RoboDK station: Assistive_UR5e.rdk

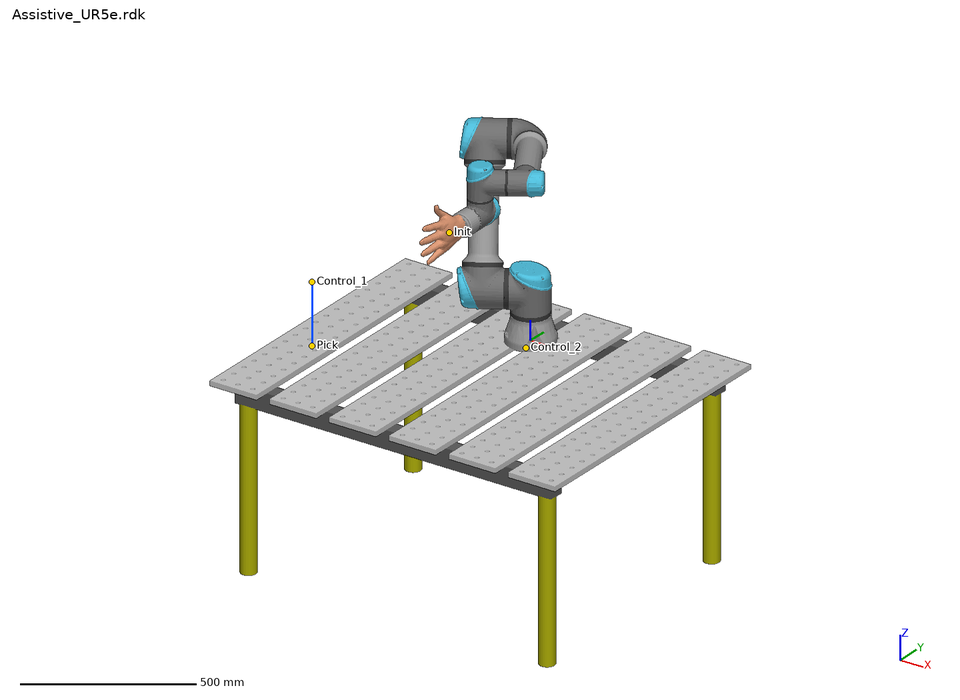
[picture v0: the station drawn from its stored meshes, robots at their saved joint values, targets as dots, program paths as lines]
Station Assistive_UR5e_SW (saved by RoboDK 5.9.2). Poses are relative to the parent item; angles as X-Y-Z fixed-axis rotations.
  - frame UR5e Base at (0, 0, 0) mm
    - robot UR5e: 6 axes, payload 5 kg, reach 850 mm, repeatability 0.03 mm, weight 18.4 kg
        modified DH rows (alpha deg, a mm, theta deg, d mm): 0, 0, 0, 162.5; 90, 0, 180, 0; 0, 425, 0, 0; 0, 392.25, 0, 133.3; -90, 0, 0, 99.7; 90, 0, 180, 99.6
        joint limits [-360, -360, -360, -360, -360, -360] to [360, 360, 360, 360, 360, 360]; home [0, -90, -90, 0, 90, 0]; saved at [-57.836, -65.392, -107.167, 172.559, -57.836, 0]
      - tool Hand, TCP at (0, 0, 50) mm, size 54.8 x 155.9 x 193.5 mm, geometry from Hand.stl
  - frame World at (0, 0, 0) mm
    - object Table at (0, 0, 0) mm, size 1193.8 x 965.2 x 609.6 mm, geometry from welding_table.sld
    - target Init (Cartesian target) at (0, -400, 500) mm, rotated rx 90 ry 0 rz 0 deg; joints [-57.836, -65.392, -107.167, 172.559, -57.836, 0] of UR5e
    - target Control_1 (joint target) at (-370, -550, 300) mm, rotated rx 90 ry -85.28 rz 0 deg; joints [-118.588, -113.226, -89.788, -156.986, -118.588, 85.275] of UR5e
    - target Pick (joint target) at (-370, -550, 100) mm, rotated rx 90.01 ry -85.28 rz -0.01 deg; joints [-118.588, -129.044, -99.259, -131.698, -118.588, 85.275] of UR5e
    - target Control_2 (joint target) at (370, -550, 300) mm, rotated rx 90.01 ry -85.28 rz -0.01 deg; joints [-33.107, -113.226, -89.788, -156.987, -33.108, 85.277] of UR5e
    - target Show (joint target) at (370, -550, 300) mm, rotated rx 90.01 ry 87.37 rz 0.01 deg; joints [-33.107, -113.226, -89.788, -156.987, -33.108, -87.373] of UR5e
  - program Init (3 instructions, listed below)
  - program Pick_object (6 instructions, listed below)
  - program Show_object (4 instructions, listed below)
  - program MainProgram (4 instructions, listed below)
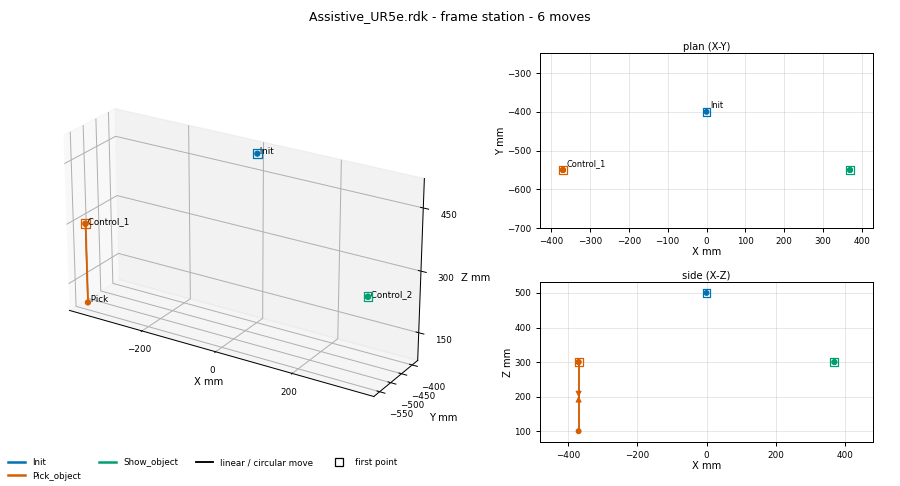
[picture p0: tool path of Assistive_UR5e.rdk in frame station, 6 of 6 moves have a stored position in this frame; points joined in program order, loops and branches not executed]

--- program Init (robot UR5e) ---
  Est. Ref.: UR5e Base
  Est. herr: Hand
  MoveJ (Init)

--- program Pick_object (robot UR5e) ---
  Est. Ref.: UR5e Base
  Est. herr: Hand
  MoveL (Control_1)
  MoveL (Pick)
  Pausa 1.0 s
  MoveL (Control_1)

--- program Show_object (robot UR5e) ---
  Est. Ref.: UR5e Base
  Est. herr: Hand
  MoveL (Control_2)
  MoveL (Show)

--- program MainProgram (robot UR5e) ---
  Llamar Init
  Llamar Pick_object
  Llamar Show_object
  Llamar Init
